(*
SPDX-FileCopyrightText: © 2026 Oleksandr Tiutyk <trofimich@gmail.com>
SPDX-License-Identifier: MIT
License: https://opensource.org/license/mit
*)

(*!
<summary>Holds at most 255 flattened entries. Inner exception graphs must be acyclic.</summary>
<description>
Input graphs must already be acyclic, including graphs from custom implementations. AddInnerException rejects
paths back to this instance before adding any entries, using a StandardException without an inner cause.
Stored entries and GetInnerException use read-only views; ownership remains with the task memory manager. Root
lookup returns a borrowed read-only view of the first entry's root, or this instance when empty. ToError
copies the aggregate message and the first entry's deepest cause into one ERROR, using the aggregate
timestamps and caller-supplied severity. Dynamic copies are explicitly registered by Clone after construction;
plain __NEW does not transfer ownership to the task manager.
</description>
*)

{attribute 'enable_dynamic_creation'}
{attribute 'no_explicit_call' := 'do not call this function block directly'}
FUNCTION_BLOCK AggregateException EXTENDS Exception IMPLEMENTS IAggregateException
VAR_STAT
	//! <summary>Class name shared by all instances of this function block.</summary>
	{attribute 'hide'} 
	_ClassName : STRING := __POUNAME();
END_VAR
VAR
	_InnerExceptions : POINTER TO IReadOnlyException;
	{attribute 'hide'} 
	_InnerExceptionCount : UINT;
END_VAR
VAR CONSTANT
	MAX_INNER_EXCEPTION_COUNT : UINT := 255;
END_VAR

(*!
<summary>Flattens aggregates; borrows dynamic inners and clones static inners for automatic cleanup.</summary>
<description>
Owns only the reference array. Accepts read-only causes; static inputs are cloned and dynamic inputs are
borrowed without exposing Clear. Allocation failure uses the shared fatal memory latch. The supplied graph
must already be acyclic, including graphs from custom implementations. The entire input graph is searched
before adding entries. A path back to this instance raises StandardException without changing this instance.
Validation follows IGeneralException and IAggregateException edges; inputs must remain live and stable during
traversal. Shared causes in separate branches are allowed. Null/empty aggregate inputs add nothing. Exceeding
255 entries raises latched OUT_OF_MEMORY before preparing the next entry. After graph validation, flattening
is incremental: prior successful additions are not rolled back on allocation or cloning failure.
</description>
*)

METHOD AddInnerException
VAR_INPUT
	innerException : IReadOnlyException; 
END_VAR
VAR
	aggregateException : IAggregateException;
	i : DINT;
	
	newInnerExceptionArray : POINTER TO IReadOnlyException;
	preparedInnerException : IReadOnlyException;

END_VAR
IF innerException = 0 THEN
	RETURN;
END_IF

IF NOT Exceptions.CanAttachInnerException(ownerException := THIS^, innerException := innerException) THEN
	Exceptions.ThrowStandard(
		sourceNamespaceName := CurrentNamespace.Name,
		sourceClassName := 'AggregateException',
		sourcePOUName := 'AddInnerException',
		sourcePosition := '',
		message := "Cannot attach an exception graph containing its prospective owner.");
END_IF

IF __QUERYINTERFACE(innerException, aggregateException) THEN
	FOR i := 0 TO TO_DINT(aggregateException.InnerExceptionCount) - 1 DO
		AddInnerException(innerException := aggregateException.GetInnerException(index := i));
	END_FOR
ELSE
	IF _InnerExceptionCount >= MAX_INNER_EXCEPTION_COUNT THEN
		DynamicMemoryManager.RaiseAllocationFailure();
	END_IF

	// Prepare the inner before replacing any existing array storage.
	IF innerException.IsDynamicInstance THEN
		preparedInnerException := innerException;
	ELSE
		__QUERYINTERFACE(innerException.Clone(), preparedInnerException);
	END_IF

	newInnerExceptionArray := __NEW(POINTER TO IReadOnlyException, (_InnerExceptionCount + 1));

	IF newInnerExceptionArray = 0 THEN
		DynamicMemoryManager.RaiseAllocationFailure();
	END_IF
		
	IF _InnerExceptionCount > 0 THEN
		Tc2_System.MEMCPY(
			destAddr := newInnerExceptionArray,
			srcAddr := _InnerExceptions,
			n := TO_UDINT(XSIZEOF(POINTER TO IReadOnlyException) * _InnerExceptionCount)
		);	
	
		__DELETE(_InnerExceptions);
	END_IF
		
	newInnerExceptionArray[_InnerExceptionCount] := preparedInnerException;
	
	_InnerExceptions := newInnerExceptionArray; 
	_InnerExceptionCount := _InnerExceptionCount + 1;
END_IF
END_METHOD

{attribute 'monitoring' := 'call'}
PROPERTY ClassName : REFERENCE TO STRING
GET
ClassName REF= _ClassName;
END_GET
END_PROPERTY

(*!
<summary>Releases the owned reference array and resets metadata; does not delete borrowed inners.</summary>
<description>
Resets the entry count, source and timestamps. Repeated Clear is allowed. Does not delete the exception
instance or unregister it from task cleanup. Other aggregates and clones borrowing the same causes remain
valid until their task cleanup. An attached dynamic cause must not be cleared through an alias.
</description>
*)

METHOD Clear
IF _InnerExceptions <> 0 THEN
	__DELETE(_InnerExceptions);
END_IF

_InnerExceptionCount := 0;

SUPER^.Clear();
END_METHOD

(*!
<summary>Returns a distinct auto-disposed aggregate with copied metadata and its own reference array.</summary>
<description>
Empty aggregates also produce a distinct empty clone. Copies source metadata and timestamps; entries retain
their order and their prepared dynamic causes remain shared. The task memory manager owns the clone until
cleanup; callers must not delete or adopt it. Clearing the source aggregate does not clear the clone or its
causes. Allocation failure uses the shared terminal memory mechanism. Descendants with additional payload must
override Clone to preserve that payload and their concrete type. Registers the newly constructed instance
before copying payload, outside FB_init. Registration failure releases the unregistered instance and raises a
terminal error; copy failure leaves the registered instance owned by the task manager for cleanup. Custom
overrides must follow the same ownership sequence.
</description>
*)

METHOD Clone : IObject
VAR
	exceptionClone : POINTER TO AggregateException;
END_VAR
exceptionClone := __NEW(AggregateException);

IF exceptionClone = 0 THEN
	DynamicMemoryManager.RaiseAllocationFailure();
END_IF

DynamicMemoryManager.RegisterAutoDisposedObject(autoDisposedObject := exceptionClone^);

exceptionClone^.CopyFields(sourceException := THIS^);

Clone := exceptionClone^;
END_METHOD

(*!
<summary>Copies aggregate metadata and entries into a distinct empty destination.</summary>
<description>
Destination must be empty and distinct from source. This helper does not clear existing entries. Source and
its causes must remain live during copying. Copies metadata and adds source entries using AddInnerException's
ownership rules; does not transfer ownership or extend cause lifetime. Copying is incremental, without
rollback on allocation or cloning failure.
</description>
*)

METHOD PROTECTED CopyFields
VAR_IN_OUT CONSTANT
	sourceException : AggregateException;	
END_VAR
VAR
	i : DINT;
END_VAR
_SourceFullPOUName := sourceException.SourceFullPOUName;
_SourcePosition := sourceException.SourcePosition;
_LocalTimestamp := sourceException.LocalTimestamp;	
_UtcTimestamp := sourceException.UtcTimestamp;	

FOR i := 0 TO TO_DINT(sourceException.InnerExceptionCount) - 1 DO
	AddInnerException(innerException := sourceException.GetInnerException(index := i));
END_FOR
END_METHOD

(*!
<summary>Reports whether the aggregate has no entries.</summary>
<description>
Equivalent to a zero immediate-entry count; does not inspect whether individual entries are empty.
</description>
*)
{attribute 'monitoring' := 'call'}
PROPERTY Empty : BOOL
GET
Empty := _InnerExceptionCount = 0;
END_GET
END_PROPERTY

(*!
<summary>Clears the aggregate during destruction.</summary>
<description>
Releases its own entry storage according to Clear. Referenced exception objects remain owned by their lifetime
manager; cleanup must not raise exceptions.
</description>
*)
//!<param name="bInCopyCode">
//! if TRUE, the exit method is called for exiting an instance that is copied afterwards (online change).
//! </param>

METHOD FB_exit : BOOL
VAR_INPUT
	
	bInCopyCode	: BOOL;
END_VAR
Clear();
END_METHOD

(*!
<summary>Returns a borrowed read-only view of an entry at a zero-based index.</summary>
<description>
Returns null for an index outside the stored range. Does not clone or transfer ownership, and does not extend
the entry lifetime beyond its task cleanup. The view is not an immutable snapshot; modifying an attached
dynamic cause through another alias is forbidden. Descendants cannot replace this view of the stored aggregate
entries; entry indexing and count refer to the same internal storage.
</description>
<param name="index">Zero-based entry index.</param>
*)
METHOD FINAL GetInnerException : IReadOnlyException
VAR_INPUT
	index : DINT;
END_VAR
IF index >= 0 AND_THEN index < _InnerExceptionCount THEN
	GetInnerException := _InnerExceptions[index];
END_IF
END_METHOD

(*!
<summary>With default options an empty aggregate returns "0 aggregated exceptions".</summary>
<description>
Formats entries in their stored order. If the result exceeds ERROR_MESSAGE capacity, preserves the prefix and
ends with an ellipsis; later entries may be omitted. Formats directly into the result without heap allocation
or builders.
</description>
*)

METHOD GetMessage : ERROR_MESSAGE
VAR_INPUT
	showSource : BOOL := FALSE;
	timestampDisplayMode : TIMESTAMP_DISPLAY_MODE := TIMESTAMP_DISPLAY_MODE.HIDDEN;
END_VAR
VAR
	i : DINT;
	innerException : IReadOnlyException;
	innerExceptionMessage : ERROR_MESSAGE;
	itemIndexText : WSTRING(16);
END_VAR
WideStrings.AppendFit255(GetMessage, TO_WSTRING(_InnerExceptionCount), Exceptions.AGGREGATE_EXCEPTION_SUFFIX);

IF timestampDisplayMode <> TIMESTAMP_DISPLAY_MODE.HIDDEN THEN
	WideStrings.AppendFit255(GetMessage, Exceptions.TIME_PREFIX);
	AppendTimestampDescription(
		targetMessage := GetMessage,
		timestampDisplayMode := timestampDisplayMode,
		localTimestamp := _LocalTimestamp,
		utcTimestamp := _UtcTimestamp
	);
END_IF

IF showSource THEN
	IF sourcePosition <> '' THEN
		WideStrings.AppendFit255(
			GetMessage,
			Exceptions.SOURCE_PREFIX,
			TO_WSTRING(_SourceFullPOUName),
			Exceptions.SOURCE_POSITION_PREFIX,
			TO_WSTRING(sourcePosition)
		);
	ELSE
		WideStrings.AppendFit255(GetMessage, Exceptions.SOURCE_PREFIX, TO_WSTRING(_SourceFullPOUName));
	END_IF
END_IF

FOR i := 0 TO TO_DINT(_InnerExceptionCount) - 1 DO
	innerException := _InnerExceptions[i];
	
	innerExceptionMessage := innerException.GetMessage(showSource := showSource, timestampDisplayMode := timestampDisplayMode);
	itemIndexText := TO_WSTRING(i);
	
	WideStrings.AppendFit255(GetMessage, WideStrings.NewLine, itemIndexText, Exceptions.MESSAGE_NUMBER_SUFFIX, " ");
	WideStrings.AppendFit(targetString := GetMessage, sourceString := innerExceptionMessage);
END_FOR
END_METHOD

(*!
<summary>Returns a borrowed read-only view of the root exception.</summary>
<description>
No clone is created and ownership is not transferred. The view does not extend the exception's lifetime and
does not expose Clear.
</description>
*)

METHOD FINAL GetRootException : IReadOnlyException
IF _InnerExceptionCount > 0 THEN
	GetRootException := GetInnerException(index := 0);
	
	GetRootException := GetRootException.GetRootException();
ELSE
	GetRootException := THIS^;
END_IF
END_METHOD

(*!
<summary>Returns the number of immediate exceptions in the aggregate.</summary>
<description>
Counts direct entries, not recursively nested causes. The aggregate supports at most 255 entries. Descendants
cannot replace this view of the stored aggregate entries; entry indexing and count refer to the same internal
storage.
</description>
*)
{attribute 'monitoring' := 'call'}
PROPERTY FINAL InnerExceptionCount : UINT
GET
InnerExceptionCount := _InnerExceptionCount;
END_GET
END_PROPERTY

(*!
<summary>Provides the library namespace used in diagnostics.</summary>
<description>
Borrowed read-only reference to the compiler-initialized library namespace; no ownership transfer.
</description>
*)
{attribute 'monitoring' := 'call'}
PROPERTY NamespaceName : REFERENCE TO STRING
GET
NamespaceName REF= CurrentNamespace.Name;
END_GET
END_PROPERTY

(*!
<summary>Reports the byte size of this concrete instance.</summary>
<description>
Uses XSIZEOF on the instance. Does not include separately allocated payloads or prove that an arbitrary
address is valid.
</description>
*)
{attribute 'monitoring' := 'call'}
PROPERTY SelfSize : ULINT
GET
SelfSize := XSIZEOF(THIS^);
END_GET
END_PROPERTY

(*!
<summary>Throws a task-managed snapshot of the aggregate exception.</summary>
<description>
Sets the supplied source metadata and current local and UTC timestamps, then delegates to
ExceptionManager.Throw. The original aggregate remains caller-owned; the registered snapshot is valid only
until task cleanup. Requires a cyclic task and follows the terminal allocation-failure policy.
</description>
*)
METHOD Throw
VAR_INPUT
	sourceNamespaceName : STRING;
	sourceClassName : STRING;
	sourcePOUName : STRING;
	sourcePosition : STRING;
END_VAR
_SourceFullPOUName := GetFullPOUName(
	sourceNamespaceName := sourceNamespaceName,
	sourceClassName := sourceClassName,
	sourcePOUName := sourcePOUName
);
_SourcePosition := sourcePosition;
_LocalTimestamp := System.SystemLocalDateTime;
_UtcTimestamp := System.SystemUtcDateTime;

ExceptionManager.Throw(exception := THIS^);
END_METHOD

(*!
<summary>Copies aggregate diagnostics and the first branch's root cause into one ERROR.</summary>
<description>
The overall message describes all entries within the GetMessage length limit. Root message and source come
from GetRootException, following the first entry to its deepest cause. Uses this aggregate's timestamps and
the supplied severity. Copies diagnostic values without transferring exception ownership. An empty aggregate
produces an explicit empty-aggregate description and no root message. An invalid target reference is ignored.
Computed diagnostic strings are held in local buffers for the duration of the receiving call.
</description>
<param name="targetError">Destination whose diagnostic fields are replaced.</param>
<param name="severity">Severity assigned to the resulting ERROR.</param>
*)
METHOD ToError
VAR_IN_OUT CONSTANT
	targetError : ERROR;
END_VAR
VAR_INPUT
	severity : ERROR_SEVERITY;	
END_VAR
VAR
	topSourceText : STRING(255);
	rootSourceText : STRING(255);
	topMessageText : ERROR_MESSAGE;
	rootMessageText : ERROR_MESSAGE;

	rootException : IReadOnlyException;
END_VAR
IF NOT __ISVALIDREF(targetError) THEN
	RETURN;
END_IF

IF _InnerExceptionCount <= 0 THEN
	topSourceText := GetSourceDescription();
	rootSourceText := Exceptions.UNSPECIFIED_SOURCE;

	targetError.Fill(
		severity := severity,
		topSource := topSourceText,
		rootSource := rootSourceText,
		topMessage := "Empty aggregate exception (zero inner exceptions)",
		rootMessage := "",
		localTimestamp := LocalTimestamp,
		utcTimestamp := UtcTimestamp
	);
	
	RETURN;
END_IF

rootException := GetRootException();

topSourceText := Strings.Concat255(TO_STRING(_InnerExceptionCount), ' exceptions occured');
rootSourceText := rootException.GetSourceDescription();
topMessageText := GetMessage();
rootMessageText := rootException.GetMessage();

targetError.Fill(
	severity := severity,
	topSource := topSourceText,
	rootSource := rootSourceText,
	topMessage := topMessageText,
	rootMessage := rootMessageText,
	localTimestamp := LocalTimestamp,
	utcTimestamp := UtcTimestamp
);
END_METHOD

END_FUNCTION_BLOCK

(* stored: Version 1.1.0.1
   POU AggregateException: Id {8695c106-e7fb-42e2-9023-16f2aac84192}, SpecialFunc None
   Folder Service members: Id {c31ba568-bfb3-4fae-ac77-198d7130e4aa}
   Method AddInnerException: Id {bfce23ea-1373-4ba3-866d-7d8a69bbfdab}
   Property ClassName: Id {bd878664-be6a-49ac-98d9-c91ba460da65}
   Get Get: Id {998929b6-4b31-437f-a5e5-a39dd1d6dc61}
   Method Clear: Id {e4a1b8c7-9686-4ca1-8667-c1a80c4453a6}
   Method Clone: Id {486d4ff9-908c-48b8-a667-acc4326b9c0c}
   Method CopyFields: Id {0584c9e4-cd70-4feb-b915-e7d77badfcc1}
   Property Empty: Id {d2ade75f-e0d1-434c-8840-7186cc0e6f7a}
   Get Get: Id {c0b1f376-6cae-43f3-86ac-6339a2e458c0}
   Method FB_exit: Id {56b27e89-e503-4505-9d3d-a810a3015a78}
   Method GetInnerException: Id {208441ce-95c7-4cde-b727-858df1415649}
   Method GetMessage: Id {76c9ffdd-6b67-4a44-aa6c-571f736f1a93}
   Method GetRootException: Id {3947d49e-1dd5-493f-96aa-4bb6602d0186}
   Property InnerExceptionCount: Id {734e1c9b-9746-493a-8ce4-7a56d60ff952}
   Get Get: Id {d38858e5-3bfc-4ef7-a005-fb8d5b223e97}
   Property NamespaceName: Id {494a86d9-380f-42f2-920d-5159f570a5a6}
   Get Get: Id {d3864769-88da-4cdf-9783-f994cd245ebc}
   Property SelfSize: Id {174b7a67-11f4-4a03-a1cf-384fffd912fd}
   Get Get: Id {0f74268c-6818-41c3-9fc5-eec449ba75e8}
   Method Throw: Id {1b8b1f86-dba3-4290-8289-61d8dd5d28c8}
   Method ToError: Id {d4ff76fe-085d-4302-a17b-b20e40bfa8ce} *)
